// TIA Portal project "1905391_000_005" (V16)

(* hardware
DEVICE "S7-1200 station_1"  S7-1200 Station
   slot 0: "Rack_0"  S7-1200 Rack  Rack  V1.0
   slot 1: "PLC_1"  CPU 1211C DC/DC/DC  6ES7 211-1AE40-0XB0  V4.4
DEVICE "HMI_1"  TP900 Comfort
   slot 0: "HMI_1"  TP900 Comfort  6AV2 124-0JC01-0AX0  16.0.0.0
   slot 1: "HMI_RT_1"  TP900 Comfort  6AV2 124-0JC01-0AX0  16.0.0.0
   slot 5: "HMI_1.IE_CP_1"  PROFINET Interface  16.0.0.0
      slot 1: "PROFINET Interface_1"  PROFINET Interface
         slot 1: "Port_1"  Port
         slot 2: "Port_2"  Port
   slot 7: "HMI_1.MPI/DP_CP_1"  MPI/DP Interface  16.0.0.0
*)

// ===== PLC "PLC_1"  CPU 1211C DC/DC/DC =====

VAR_GLOBAL   // PLC tag table "Default tag table"
   "System_Byte" AT %MB1 : Byte;
   "FirstScan" AT %M1.0 : Bool;
   "DiagStatusUpdate" AT %M1.1 : Bool;
   "AlwaysTRUE" AT %M1.2 : Bool;
   "AlwaysFALSE" AT %M1.3 : Bool;
   "Clock_Byte" AT %MB0 : Byte;
   "Clock_10Hz" AT %M0.0 : Bool;
   "Clock_5Hz" AT %M0.1 : Bool;
   "Clock_2.5Hz" AT %M0.2 : Bool;
   "Clock_2Hz" AT %M0.3 : Bool;
   "Clock_1.25Hz" AT %M0.4 : Bool;
   "Clock_1Hz" AT %M0.5 : Bool;
   "Clock_0.625Hz" AT %M0.6 : Bool;
   "Clock_0.5Hz" AT %M0.7 : Bool;
END_VAR

VAR_GLOBAL CONSTANT   // PLC tag table "Default tag table"
   "STRING_LENGTH" : Int := 20;
   "ADP_PARAMETER_LENGTH" : Int := 5;
   "NULL_TOKEN" : Int := -1;
END_VAR

TYPE "Database.UDT"
   STRUCT
      elements : "Elements.Data.UDT";
      wires : "Wires.Data.UDT";
   END_STRUCT;
END_TYPE

TYPE "Divider.UDT"
   STRUCT
      background_animate : Int;
      background_visible : Bool;
      line_animate : Int;
      line_visible : Bool;
   END_STRUCT;
END_TYPE

TYPE "Row_Data.UDT"
   STRUCT
      background_animate : Int;
      background_visible : Bool;
      cell_0_animate : Int;
      cell_0_value : String[50];
      cell_0_visible : Bool;
      cell_1_animate : Int;
      cell_1_enable : Bool;
      cell_1_input_finished : Bool;
      cell_1_value : String[50];
      cell_1_visible : Bool;
   END_STRUCT;
END_TYPE

TYPE "Row_Label.UDT"
   STRUCT
      background_animate : Int;
      background_visible : Bool;
      cell_0_animate : Int;
      cell_0_value : String[50];
      cell_0_visible : Bool;
      cell_1_animate : Int;
      cell_1_value : String[50];
      cell_1_visible : Bool;
   END_STRUCT;
END_TYPE

TYPE "HMI_Interface.UDT"
   STRUCT
      elements : "Elements.HMI.UDT";
      wires : "Wires.HMI.UDT";
   END_STRUCT;
END_TYPE

TYPE "LED_Interface.UDT"
   STRUCT
      elements : "Elements.LED.UDT";
      wires : "Wires.LED.UDT";
   END_STRUCT;
END_TYPE

TYPE "Navigation.UDT"
   STRUCT
      material_actuate : Bool;
      material_animate : Int;
      material_cover_visible : Bool;
      wire_actuate : Bool;
      wire_animate : Int;
      wire_cover_visible : Bool;
   END_STRUCT;
END_TYPE

TYPE "Row_Custom.UDT"
   STRUCT
      background_animate : Int;
      background_visible : Bool;
      cell_0_animate : Int;
      cell_0_enable : Bool;
      cell_0_input_finished : Bool;
      cell_0_value : String[50];
      cell_0_visible : Bool;
      cell_1_animate : Int;
      cell_1_enable : Bool;
      cell_1_input_finished : Bool;
      cell_1_value : String[50];
      cell_1_visible : Bool;
   END_STRUCT;
END_TYPE

// folder: ADP Data

TYPE "ADP.Row.2_Cells.UDT"
   STRUCT
      me : Array[0..1] of "ADP.Cell.UDT";
   END_STRUCT;
END_TYPE

TYPE "ADP.Cell.UDT"
   STRUCT
      color : String["ADP_PARAMETER_LENGTH"];
      flashing : String["ADP_PARAMETER_LENGTH"];
      h_align : String["ADP_PARAMETER_LENGTH"];
      lince_control : String["ADP_PARAMETER_LENGTH"];
      scroll_speed : String["ADP_PARAMETER_LENGTH"];
      size_and_face : String["ADP_PARAMETER_LENGTH"];
      v_align : String["ADP_PARAMETER_LENGTH"];
      value : String["STRING_LENGTH"];
   END_STRUCT;
END_TYPE

TYPE "ADP.Message_Buffer.UDT"
   STRUCT
      me : Array[0..999] of Byte;
   END_STRUCT;
END_TYPE

TYPE "ADP.Decoded.UDT"
   STRUCT
      color : "ADP.Decoded.Color.UDT";
      flash : "ADP.Decoded.Flash.UDT";
      horizontal_alignment : "ADP.Decoded.Horizontal_Alignment.UDT";
      line_control : "ADP.Decoded.Line_Control.UDT";
      scroll_speed : "ADP.Decoded.Scroll_Speed.UDT";
      size_and_face : "ADP.Decoded.Size_and_Face.UDT";
      vertical_alignment : "ADP.Decoded.Vertical_Alignment.UDT";
   END_STRUCT;
END_TYPE

TYPE "ADP.Decoded.Color.UDT"
   STRUCT
      black : String[8] := 'black';
      blue : String[8] := 'blue';
      green : String[8] := 'green';
      mix_1 : String[8] := 'mix 1';
      mix_2 : String[8] := 'mix 2';
      mix_3 : String[8] := 'mix 3';
      mix_4 : String[8] := 'mix 4';
      red : String[8] := 'red';
      white : String[8] := 'white';
      yellow : String[8] := 'yellow';
   END_STRUCT;
END_TYPE

TYPE "ADP.Decoded.Flash.UDT"
   STRUCT
      off : String[8] := 'off';
      on : String[8] := 'on';
   END_STRUCT;
END_TYPE

TYPE "ADP.Decoded.Horizontal_Alignment.UDT"
   STRUCT
      center : String[8] := 'center';
      left : String[8] := 'left';
      right : String[8] := 'right';
   END_STRUCT;
END_TYPE

TYPE "ADP.Encoded.UDT"
VERSION : 0.1
   STRUCT
      file_system : "ADP.Encoded.File_System.UDT";
      formatting : "ADP.Encoded.Formatting.UDT";
   END_STRUCT;
END_TYPE

TYPE "ADP.Message_Formats.Encoded.UDT"
   STRUCT
      color : String [5];
      flash : String [5];
      scroll_speed : String [5];
      size_and_face : String [5];
      vertical_alignment : String [5];
      horizontal_alignment : String [5];
   END_STRUCT;
END_TYPE

TYPE "ADP.Message_Formats.Decoded.UDT"
   STRUCT
      color : String [20];
      flash : String [20];
      scroll_speed : String [20];
      size_and_face : String [20];
      vertical_alignment : String [20];
      horizontal_alignment : String [20];
   END_STRUCT;
END_TYPE

TYPE "ADP.Decoded.Scroll_Speed.UDT"
   STRUCT
      slowest : String[9] := 'slowest';
      slow : String[9] := 'slow';
      normal : String[9] := 'normal';
      fast : String[9] := 'fast';
      fastest : String[9] := 'fastest';
   END_STRUCT;
END_TYPE

TYPE "ADP.Decoded.Size_and_Face.UDT"
   STRUCT
      bold_5 : String[11] := 'bold 5';
      bold_11 : String[11] := 'bold 11';
      bold_14 : String[11] := 'bold 14';
      bold_15 : String[11] := 'bold 15';
      bold_16 : String[11] := 'bold 16';
      bold_22 : String[11] := 'bold 22';
      bold_30 : String[11] := 'bold 30';
      bold_32 : String[11] := 'bold 32';
      bold_40 : String[11] := 'bold 40';
      normal_5 : String[11] := 'normal 5';
      normal_7 : String[11] := 'normal 7';
      normal_9 : String[11] := 'normal 9';
      normal_11 : String[11] := 'normal 11';
      normal_14 : String[11] := 'normal 14';
      normal_15 : String[11] := 'normal 15';
      normal_16 : String[11] := 'normal 16';
      normal_22 : String[11] := 'normal 22';
      normal_24 : String[11] := 'normal 24';
      normal_30 : String[11] := 'normal 30';
      normal_32 : String[11] := 'normal 32';
      normal_40 : String[11] := 'normal 40';
   END_STRUCT;
END_TYPE

TYPE "ADP.Decoded.Vertical_Alignment.UDT"
   STRUCT
      bottom_hold : String[15] := 'bottom hold';
      fill_hold : String[15] := 'fill hold';
      middle_hold : String[15] := 'middle hold';
      top_hold : String[15] := 'top hold';
      bottom_scroll : String[15] := 'bottom scroll';
      fill_scroll : String[15] := 'fill scroll';
      middle_scroll : String[15] := 'middle scroll';
      top_scroll : String[15] := 'top scroll';
   END_STRUCT;
END_TYPE

TYPE "ADP.Encoded.File_System.UDT"
   STRUCT
      "00 Start of Header" : String[5] := '$01';
      "01 Address" : String[5] := 'Z00';
      "02 Start of Text" : String[5] := '$02';
      "03 Command & File" : String[5] := 'AA';
      "04 END" : String[5] := '$04';
   END_STRUCT;
END_TYPE

TYPE "ADP.Encoded.Formatting.UDT"
   STRUCT
      color : "ADP.Encoded.Formatting.Color.UDT";
      flashing : "ADP.Encoded.Formatting.Flashing.UDT";
      horizontal_alignment : "ADP.Encoded.Formatting.Horizonta_Alignment.UDT";
      line_control : "ADP.Encoded.Formatting.Line_Control.UDT";
      scroll_speed : "ADP.Encoded.Formatting.Scroll_Speed.UDT";
      size_and_face : "ADP.Encoded.Formatting.Size_and_Face.UDT";
      vertical_alignment : "ADP.Encoded.Formatting.Vertical_Alignment.UDT";
   END_STRUCT;
END_TYPE

TYPE "ADP.Encoded.Formatting.Color.UDT"
   STRUCT
      black : String[5] := '$1C0';
      blue : String[5] := '$1C8';
      green : String[5] := '$1C2';
      mix_1 : String[5] := '$1C4';
      mix_2 : String[5] := '$1C5';
      mix_3 : String[5] := '$1C6';
      mix_4 : String[5] := '$1CY';
      red : String[5] := '$1C1';
      white : String[5] := '$1C9';
      yellow : String[5] := '$1C3';
   END_STRUCT;
END_TYPE

TYPE "ADP.Encoded.Formatting.Flashing.UDT"
   STRUCT
      off : String[5] := '$070';
      on : String[5] := '$071';
   END_STRUCT;
END_TYPE

TYPE "ADP.Encoded.Formatting.Size_and_Face.UDT"
   STRUCT
      bold_5 : String[5] := '$1AG';
      bold_11 : String[5] := '$1AH';
      bold_14 : String[5] := '$1A5';
      bold_15 : String[5] := '$1A6';
      bold_16 : String[5] := '$1A7';
      bold_22 : String[5] := '$1AC';
      bold_30 : String[5] := '$1AI';
      bold_32 : String[5] := '$1AJ';
      bold_40 : String[5] := '$1AK';
      normal_5 : String[5] := '$1A0';
      normal_7 : String[5] := '$1A1';
      normal_9 : String[5] := '$1A8';
      normal_11 : String[5] := '$1A9';
      normal_14 : String[5] := '$1A2';
      normal_15 : String[5] := '$1A3';
      normal_16 : String[5] := '$1A4';
      normal_22 : String[5] := '$1AA';
      normal_24 : String[5] := '$1AB';
      normal_30 : String[5] := '$1AD';
      normal_32 : String[5] := '$1AE';
      normal_40 : String[5] := '$1AF';
   END_STRUCT;
END_TYPE

TYPE "ADP.Encoded.Formatting.Horizonta_Alignment.UDT"
   STRUCT
      center : String[5] := '$L1';
      left : String[5] := '$L0';
      right : String[5] := '$L2';
   END_STRUCT;
END_TYPE

TYPE "ADP.Encoded.Formatting.Vertical_Alignment.UDT"
   STRUCT
      middle_hold : String[5] := '$1B b';
      fill_hold : String[5] := '$1B"b';
      bottom_hold : String[5] := '$1B&b';
      top_hold : String[5] := '$1B0b';
      bottom_scroll : String[5] := '$1B a';
      fill_scroll : String[5] := '$1B"a';
      middle_scroll : String[5] := '$1B&a';
      top_scroll : String[5] := '$1B0a';
   END_STRUCT;
END_TYPE

TYPE "ADP.Encoded.Formatting.Scroll_Speed.UDT"
   STRUCT
      slowest : String[5] := '$15';
      slow : String[5] := '$16';
      normal : String[5] := '$17';
      fast : String[5] := '$18';
      fastest : String[5] := '$19';
   END_STRUCT;
END_TYPE

TYPE "ADP.Encoded.Formatting.Line_Control.UDT"
   STRUCT
      new_line : String[5] := '$R';
      word_wrap : String[5] := '';
   END_STRUCT;
END_TYPE

TYPE "ADP.Decoded.Line_Control.UDT"
   STRUCT
      new_line : String[9] := 'new line';
      word_wrap : String[9] := 'word wrap';
   END_STRUCT;
END_TYPE

// folder: Element Data

TYPE "Elements.HMI.UDT"
   STRUCT
      chromium : "Row.(IOF.String_IOF.Real).UDT";
      custom : "Row.(IOF.String_IOF.Real).UDT";
      header : "Row.(IOF.String_IOF.String).UDT";
      heat : "Row.(IOF.String_IOF.Real).UDT";
      manganese : "Row.(IOF.String_IOF.Real).UDT";
      molybdenum : "Row.(IOF.String_IOF.Real).UDT";
      nickel : "Row.(IOF.String_IOF.Real).UDT";
      silicon : "Row.(IOF.String_IOF.Real).UDT";
      vanadium : "Row.(IOF.String_IOF.Real).UDT";
   END_STRUCT;
   // header.cell_00.value := 'Material';
   // header.cell_01.value := 'Bags';
END_TYPE

TYPE "Elements.Data.UDT"
   STRUCT
      chromium : Real;
      custom_value : Real;
      custom_name : String[50];
      heat : Real;
      manganese : Real;
      molybdenum : Real;
      nickel : Real;
      silicon : Real;
      vanadium : Real;
   END_STRUCT;
END_TYPE

TYPE "Elements.LED.UDT"
   STRUCT
      chromium : "ADP.Row.2_Cells.UDT";
      custom : "ADP.Row.2_Cells.UDT";
      header : "ADP.Row.2_Cells.UDT";
      heat : "ADP.Row.2_Cells.UDT";
      manganese : "ADP.Row.2_Cells.UDT";
      molybdenum : "ADP.Row.2_Cells.UDT";
      nickel : "ADP.Row.2_Cells.UDT";
      silicon : "ADP.Row.2_Cells.UDT";
      vanadium : "ADP.Row.2_Cells.UDT";
   END_STRUCT;
   // chromium.me[0].value := 'chromium';
   // heat.me[0].value := 'heat';
   // manganese.me[0].value := 'manganese';
   // molybdenum.me[0].value := 'molybdenum';
   // nickel.me[0].value := 'nickel';
   // silicon.me[0].value := 'silicon';
   // vanadium.me[0].value := 'vanadium';
   // custom.me[0].value := 'Custom';
   // header.me[0].value := 'Material';
   // header.me[1].value := 'Bags';
END_TYPE

// folder: Wire Data

TYPE "Wire.UDT"
   STRUCT
      aluminum : Real;
      calcium_silicon : Real;
      carbon : Real;
      custom : Real;
      heat : Real;
      sulfur : Real;
   END_STRUCT;
END_TYPE

TYPE "Wires.LED.UDT"
   STRUCT
      aluminum : "ADP.Row.2_Cells.UDT";
      calcium_silicon : "ADP.Row.2_Cells.UDT";
      carbon : "ADP.Row.2_Cells.UDT";
      custom : "ADP.Row.2_Cells.UDT";
      heat : "ADP.Row.2_Cells.UDT";
      sulfur : "ADP.Row.2_Cells.UDT";
   END_STRUCT;
   // aluminum.me[0].value := 'AL Wire';
   // calcium_silicon.me[0].value := 'Cal/Sil Wire';
   // carbon.me[0].value := 'Carbon Wire';
   // heat.me[0].value := 'HEAT';
   // sulfur.me[0].value := 'Sulfur Wire';
   // custom.me[0].value := 'Custom';
END_TYPE

TYPE "Wire.HMI.UDT"
   STRUCT
      aluminum : "Row_Data.UDT";
      bottom_border : "Divider.UDT";
      calcium_silicon : "Row_Data.UDT";
      carbon : "Row_Data.UDT";
      divider : "Divider.UDT";
      header : "Row_Data.UDT";
      heat : "Row_Data.UDT";
      sulfur : "Row_Data.UDT";
   END_STRUCT;
END_TYPE

// folder: data

DATA_BLOCK "Database.Data"   // DB1
{ S7_Optimized_Access := 'TRUE' }
VERSION : 0.1
BEGIN
END_DATA_BLOCK

// folder: display/HMI

DATA_BLOCK "HMI_Interface.Data"   // DB2
{ S7_Optimized_Access := 'TRUE' }
VERSION : 0.1
BEGIN
END_DATA_BLOCK

// folder: display/LED

DATA_BLOCK "LED_Interface.Data"   // DB3
{ S7_Optimized_Access := 'TRUE' }
VERSION : 0.1
BEGIN
END_DATA_BLOCK

// folder: (top level)

FUNCTION "Row_Data.Background.Animate" : Void   // FC1, SCL
{ S7_Optimized_Access := 'TRUE' }
VERSION : 0.1
   VAR_IN_OUT
      background : Int;
   END_VAR
BEGIN
END_FUNCTION

FUNCTION "Strip_Sign" : String   // FC20, SCL
{ S7_Optimized_Access := 'TRUE' }
VERSION : 0.1
   VAR_INPUT
      "string" : String;
   END_VAR
   VAR_TEMP
      Length : Int;
      "String Box" : String;
      "Test Character" : String;
   END_VAR
   VAR CONSTANT
      "+" : Char := '+';
      "-" : Char := '-';
   END_VAR
BEGIN
   #"String Box" := #string;
   #"Test Character" := LEFT_STRING(IN := #"String Box",
                                    L := 1);
   IF #"Test Character" = #"+" OR #"Test Character" = #"-" THEN
       #Length := LEN(#"String Box");
       #"String Box" := RIGHT_STRING(IN := #"String Box", L := #Length - 1);

   END_IF;
   #"Strip Sign" := #"String Box";
END_FUNCTION

FUNCTION "Trim" : String   // FC21, SCL
{ S7_Optimized_Access := 'TRUE' }
AUTHOR : Machado
FAMILY : String
VERSION : 1.0
// removes leading and trailing whitespace from input string
   VAR_INPUT
      "string" : String;
   END_VAR
   VAR_TEMP
      ret : String;
   END_VAR
   VAR CONSTANT
      space : String := ' ';
   END_VAR
BEGIN
   #ret := #string;
   WHILE LEFT(IN := #ret, L := 1) = #space DO
       #ret := RIGHT(IN := #ret, L := LEN(#ret) - 1);
   END_WHILE;
   WHILE RIGHT(IN := #ret, L := 1) = #space DO
       #ret := LEFT(IN := #ret, L := LEN(#ret) - 1);
   END_WHILE;
   #Trim := #ret;
END_FUNCTION

FUNCTION "Upper" : String   // FC22, SCL
{ S7_Optimized_Access := 'TRUE' }
AUTHOR : Machado
FAMILY : String
VERSION : 1.0
// returns the input string converted to all upper case
   VAR_INPUT
      "string" : String;
   END_VAR
   VAR_TEMP
      "type" : Bool;
      stringBox : String;
      status : Int;
      charArr : Array[0..255] of Char;
      cntChar : UInt;
      pChar : Int;
   END_VAR
   VAR CONSTANT
      asciiLow : Char := 'a';
      asciiHigh : Char := 'z';
      asciiCaseOffset : Int := 32;
   END_VAR
BEGIN
   Strg_TO_Chars(Strg := #string,
                 pChars := 0,
                 Cnt => #cntChar,
                 Chars := #charArr);

   FOR #pChar := 0 TO UINT_TO_INT(#cntChar) - 1 DO
       IF #asciiLow <= #charArr[#pChar] AND #charArr[#pChar] <= #asciiHigh THEN
           #charArr[#pChar] := INT_TO_CHAR(CHAR_TO_INT(#charArr[#pChar]) - #asciiCaseOffset);
       END_IF;
   END_FOR;

   Chars_TO_Strg(Chars := #charArr,
                 pChars := 0,
                 Cnt := #cntChar,
                 Strg => #stringBox);

   #Upper := #stringBox;
END_FUNCTION

ORGANIZATION_BLOCK "Main"   // OB1, LAD, ProgramCycle
TITLE = "Main Program Sweep (Cycle)"
{ S7_Optimized_Access := 'TRUE' }
VERSION : 0.1
   VAR_INPUT
      Initial_Call : Bool;   // Initial call of this OB
      Remanence : Bool;   // =True, if remanent data are available
   END_VAR
BEGIN
END_ORGANIZATION_BLOCK

// folder: display

FUNCTION_BLOCK "Display"   // FB5, SCL
{ S7_Optimized_Access := 'TRUE' }
VERSION : 0.1
BEGIN
   REGION "HMI"

   END_REGION

   REGION "LED"

   END_REGION
END_FUNCTION_BLOCK

// folder: display/HMI

FUNCTION_BLOCK "HMI"   // FB6, SCL
{ S7_Optimized_Access := 'TRUE' }
VERSION : 0.1
   VAR_IN_OUT
      interface : "HMI_Interface.UDT";
   END_VAR
   VAR
      place_holder : Bool;
   END_VAR
BEGIN
   REGION "VALIDATE INPUT"
       "HMI.Validate"();
   END_REGION


   REGION "DISPLAY VALUES"
       // may not be needed, handeled entirely in middleware
   END_REGION


   REGION "ANIMATE"
       "HMI.Animate"();
   END_REGION
END_FUNCTION_BLOCK

FUNCTION "HMI.Animate" : Void   // FC8, SCL
{ S7_Optimized_Access := 'TRUE' }
VERSION : 0.1
BEGIN
   "Element.Animate"();
   "Wire.Animate"();
END_FUNCTION

FUNCTION "HMI.Validate" : Void   // FC9, SCL
{ S7_Optimized_Access := 'TRUE' }
VERSION : 0.1
BEGIN
   "Element.Validate"();
   "Wire.Validate"();
END_FUNCTION

FUNCTION "HMI.Display" : Void   // FC10, SCL
{ S7_Optimized_Access := 'TRUE' }
VERSION : 0.1
   VAR_INPUT
      database : Bool;
   END_VAR
BEGIN
END_FUNCTION

// folder: display/HMI/Wire

FUNCTION "HMI.Animate.Wire" : Void   // FC3, SCL
{ S7_Optimized_Access := 'TRUE' }
VERSION : 0.1
   VAR_IN_OUT
      wire : "Wire.HMI.UDT";
   END_VAR
BEGIN
END_FUNCTION

FUNCTION "Wire.Animate.Aluminum" : Void   // FC4, SCL
{ S7_Optimized_Access := 'TRUE' }
VERSION : 0.1
BEGIN
END_FUNCTION

// folder: display/LED

FUNCTION_BLOCK "LED"   // FB7, SCL
{ S7_Optimized_Access := 'TRUE' }
VERSION : 0.1
   VAR
      Elements_Sign : "Elements_Sign";
      Wires_Sign : "Wires_Sign";
   END_VAR
BEGIN
   REGION "ELEMENTS"
       #Elements_Sign();
   END_REGION

   REGION "WIRES"
       #Wires_Sign();
   END_REGION
END_FUNCTION_BLOCK

FUNCTION_BLOCK "LED.Sign.Send"   // FB9, SCL
{ S7_Optimized_Access := 'TRUE' }
VERSION : 0.1
   VAR_INPUT
      data : "ADP.Message_Buffer.UDT";
      id : Conn_Ouc;
      request : Bool;
   END_VAR
   VAR
      TSEND : TSEND;
   END_VAR
BEGIN
   #TSEND(REQ := #request,
          ID := #id,
          DATA := #data);
END_FUNCTION_BLOCK

FUNCTION_BLOCK "LED.Sign"   // FB10, SCL
{ S7_Optimized_Access := 'TRUE' }
VERSION : 0.1
   VAR_INPUT
      id : Conn_Ouc;
      connection_parameters : TCON_Param;
      requests : Struct
         connect : Bool;
         diagnostics : Bool;
         disconnect : Bool;
         reset : Bool;
         send : Bool;
      END_STRUCT;
   END_VAR
   VAR
      Connect : "LED.Sign.Connect";
      Disconnect : "LED.Sign.Disconnect";
      Send : "LED.Sign.Send";
      Reset : "LED.Sign.Reset";
      Diagnostics : "LED.Sign.Diagnostics";
   END_VAR
BEGIN
   #Connect(request := #requests.connect,
            id := #id,
            connection_parameters := #connection_parameters);

   #Disconnect(id := #id,
               request := #requests.disconnect);

   #Send(id := #id,
         request := #requests.send);

   #Reset(id := #id,
          request := #requests.reset);

   #Diagnostics(id := #id,
                request := #requests.diagnostics);
END_FUNCTION_BLOCK

FUNCTION_BLOCK "LED.Sign.Connect"   // FB11, SCL
{ S7_Optimized_Access := 'TRUE' }
VERSION : 0.1
   VAR_INPUT
      request : Bool;
      id : Conn_Ouc;
      connection_parameters : TCON_Param;
   END_VAR
   VAR
      TCON : TCON;
   END_VAR
BEGIN
   #TCON(REQ := #request,
         ID := #id,
         CONNECT := #connection_parameters);
END_FUNCTION_BLOCK

FUNCTION_BLOCK "LED.Sign.Reset"   // FB12, SCL
{ S7_Optimized_Access := 'TRUE' }
VERSION : 0.1
   VAR_INPUT
      request : Bool;
      id : Conn_Ouc;
   END_VAR
   VAR
      T_RESET : T_RESET;
   END_VAR
BEGIN
   #T_RESET(REQ:=#request,
            ID:=#id,
            DONE=>_bool_out_,
            BUSY=>_bool_out_,
            ERROR=>_bool_out_,
            STATUS=>_word_out_);
END_FUNCTION_BLOCK

FUNCTION_BLOCK "LED.Sign.Disconnect"   // FB13, SCL
{ S7_Optimized_Access := 'TRUE' }
VERSION : 0.1
   VAR_INPUT
      request : Bool;
      id : Conn_Ouc;
   END_VAR
   VAR
      TDISCON : TDISCON;
   END_VAR
BEGIN
   #TDISCON(REQ := #request,
            ID := #id);
END_FUNCTION_BLOCK

FUNCTION_BLOCK "LED.Sign.Diagnostics"   // FB14, SCL
{ S7_Optimized_Access := 'TRUE' }
VERSION : 0.1
   VAR_INPUT
      request : Bool;
      id : Conn_Ouc;
   END_VAR
   VAR
      T_DIAG : T_DIAG;
   END_VAR
BEGIN
   #T_DIAG(REQ:=#request,
           ID:=#id);
END_FUNCTION_BLOCK

// folder: display/LED/Elements Sign

FUNCTION_BLOCK "Elements_Sign"   // FB16, SCL
{ S7_Optimized_Access := 'TRUE' }
VERSION : 0.1
   VAR
      Sign : "LED.Sign";
      id : Conn_Ouc;
      connection_parameters : TCON_Param;
   END_VAR
BEGIN
   "Elements_Sign.Assemble_Message"();
   #Sign(id := #id,
         connection_parameters := #connection_parameters);
END_FUNCTION_BLOCK

FUNCTION "Elements_Sign.Assemble_Message" : Void   // FC11, SCL
{ S7_Optimized_Access := 'TRUE' }
VERSION : 0.1
BEGIN
END_FUNCTION

// folder: display/LED/Wires Sign

FUNCTION_BLOCK "Wires_Sign"   // FB15, SCL
{ S7_Optimized_Access := 'TRUE' }
VERSION : 0.1
   VAR
      Sign : "LED.Sign";
      id : Conn_Ouc;
      connection_parameters : TCON_Param;
   END_VAR
BEGIN
   "Wires_Sign.Assemble_Message"();
   #Sign(id := #id,
         connection_parameters := #connection_parameters);
END_FUNCTION_BLOCK

FUNCTION "Wires_Sign.Assemble_Message" : Void   // FC12, SCL
{ S7_Optimized_Access := 'TRUE' }
VERSION : 0.1
BEGIN
END_FUNCTION

// folder: divider

FUNCTION "Divider.Show" : Void   // FC2, SCL
{ S7_Optimized_Access := 'TRUE' }
VERSION : 0.1
   VAR_IN_OUT
      divider : "Divider.UDT";
   END_VAR
   VAR CONSTANT
      MODE : Bool := TRUE;
   END_VAR
BEGIN
   #divider.background_visible := #MODE;
   #divider.line_visible := #MODE;
END_FUNCTION

FUNCTION "Divider.Hide" : Void   // FC2, SCL
{ S7_Optimized_Access := 'TRUE' }
VERSION : 0.1
   VAR_IN_OUT
      divider : "Divider.UDT";
   END_VAR
   VAR CONSTANT
      MODE : Bool := FALSE;
   END_VAR
BEGIN
   #divider.background_visible := #MODE;
   #divider.line_visible := #MODE;
END_FUNCTION

FUNCTION "Divider.Hide_Line" : Void   // FC13, SCL
{ S7_Optimized_Access := 'TRUE' }
VERSION : 0.1
   VAR_TEMP
      divider : "Divider.UDT";
   END_VAR
   VAR CONSTANT
      MODE : Bool := TRUE;
   END_VAR
BEGIN
   #divider.line_visible := #MODE;
END_FUNCTION

// folder: middleware

FUNCTION_BLOCK "Middleware"   // FB2, SCL
{ S7_Optimized_Access := 'TRUE' }
VERSION : 0.1
   VAR_IN_OUT
      database : "Database.UDT";
      hmi : "HMI_Interface.UDT";
      led : "LED_Interface.UDT";
   END_VAR
   VAR
      elements : "Elements";
      wires : "Wires";
   END_VAR
BEGIN
   #elements(database := #database.elements,
             hmi := #hmi.elements,
             led := #led.elements);

   #wires(database := #database.wires,
          hmi := #hmi.wires,
          led := #led.wires);
END_FUNCTION_BLOCK

// folder: row_data

FUNCTION "Row_Data.Animate" : Void   // FC5, SCL
{ S7_Optimized_Access := 'TRUE' }
VERSION : 0.1
   VAR_IN_OUT
      row_data : "Row_Data.UDT";
   END_VAR
BEGIN
   #row_data.background_animate := "NULL_TOKEN";
   #row_data.cell_0_animate := "NULL_TOKEN";
   #row_data.cell_1_animate := "NULL_TOKEN";
END_FUNCTION

FUNCTION "Row_Data.Show" : Void   // FC6, SCL
{ S7_Optimized_Access := 'TRUE' }
VERSION : 0.1
   VAR_IN_OUT
      row_data : "Row_Data.UDT";
   END_VAR
   VAR CONSTANT
      MODE : Bool := TRUE;
   END_VAR
BEGIN
   #row_data.background_visible := #MODE;
   #row_data.cell_0_visible := #MODE;
   #row_data.cell_1_visible := #MODE;
END_FUNCTION

FUNCTION "Row_Data.Hide" : Void   // FC6, SCL
{ S7_Optimized_Access := 'TRUE' }
VERSION : 0.1
   VAR_IN_OUT
      row_data : "Row_Data.UDT";
   END_VAR
   VAR CONSTANT
      MODE : Bool := FALSE;
   END_VAR
BEGIN
   #row_data.background_visible := #MODE;
   #row_data.cell_0_visible := #MODE;
   #row_data.cell_1_visible := #MODE;
END_FUNCTION

FUNCTION "Row_Data.Enable" : Void   // FC7, SCL
{ S7_Optimized_Access := 'TRUE' }
VERSION : 0.1
   VAR_IN_OUT
      row_data : "Row_Data.UDT";
   END_VAR
BEGIN
   #row_data.cell_1_enable := TRUE;
END_FUNCTION

// ===== library types =====

TYPE "Row.UDT"
   STRUCT
      background_animate : Int;
      background_visible : Bool;
      cell_0_animate : Int;
      cell_0_value : String[50];
      cell_0_visible : Bool;
      cell_1_animate : Int;
      cell_1_enable : Bool;
      cell_1_input_finished : Bool;
      cell_1_value : String[50];
      cell_1_visible : Bool;
   END_STRUCT;
END_TYPE

// ===== library: MasterCopy "Copy of PLC data types in ADP Data" =====

// folder: ADP Data

TYPE "ADP: Encoded"
VERSION : 0.1
   STRUCT
      file_system : "ADP: Encoded: File System";
      formatting : "ADP: Encoded: Formatting";
   END_STRUCT;
END_TYPE

TYPE "ADP: Decoded"
   STRUCT
      color : "ADP: Decoded: Color";
      flash : "ADP: Decoded: Flash";
      horizontal_alignment : "ADP: Decoded: Horizontal Alignment";
      line_control : "ADP: Decoded: Line Control";
      scroll_speed : "ADP: Decoded: Scroll Speed";
      size_and_face : "ADP: Decoded: Size and Face";
      vertical_alignment : "ADP: Decoded: Vertical Alignment";
   END_STRUCT;
END_TYPE

TYPE "ADP: Decoded: Color"
   STRUCT
      black : String[8] := 'black';
      blue : String[8] := 'blue';
      green : String[8] := 'green';
      mix_1 : String[8] := 'mix 1';
      mix_2 : String[8] := 'mix 2';
      mix_3 : String[8] := 'mix 3';
      mix_4 : String[8] := 'mix 4';
      red : String[8] := 'red';
      white : String[8] := 'white';
      yellow : String[8] := 'yellow';
   END_STRUCT;
END_TYPE

TYPE "ADP: Decoded: Flash"
   STRUCT
      off : String[8] := 'off';
      on : String[8] := 'on';
   END_STRUCT;
END_TYPE

TYPE "ADP: Decoded: Horizontal Alignment"
   STRUCT
      center : String[8] := 'center';
      left : String[8] := 'left';
      right : String[8] := 'right';
   END_STRUCT;
END_TYPE

TYPE "ADP: Message Formats: Encoded"
   STRUCT
      color : String [5];
      flash : String [5];
      scroll_speed : String [5];
      size_and_face : String [5];
      vertical_alignment : String [5];
      horizontal_alignment : String [5];
   END_STRUCT;
END_TYPE

TYPE "ADP: Message Formats: Decoded"
   STRUCT
      color : String [20];
      flash : String [20];
      scroll_speed : String [20];
      size_and_face : String [20];
      vertical_alignment : String [20];
      horizontal_alignment : String [20];
   END_STRUCT;
END_TYPE

TYPE "ADP: Decoded: Scroll Speed"
   STRUCT
      slowest : String[9] := 'slowest';
      slow : String[9] := 'slow';
      normal : String[9] := 'normal';
      fast : String[9] := 'fast';
      fastest : String[9] := 'fastest';
   END_STRUCT;
END_TYPE

TYPE "ADP: Decoded: Size and Face"
   STRUCT
      bold_5 : String[11] := 'bold 5';
      bold_11 : String[11] := 'bold 11';
      bold_14 : String[11] := 'bold 14';
      bold_15 : String[11] := 'bold 15';
      bold_16 : String[11] := 'bold 16';
      bold_22 : String[11] := 'bold 22';
      bold_30 : String[11] := 'bold 30';
      bold_32 : String[11] := 'bold 32';
      bold_40 : String[11] := 'bold 40';
      normal_5 : String[11] := 'normal 5';
      normal_7 : String[11] := 'normal 7';
      normal_9 : String[11] := 'normal 9';
      normal_11 : String[11] := 'normal 11';
      normal_14 : String[11] := 'normal 14';
      normal_15 : String[11] := 'normal 15';
      normal_16 : String[11] := 'normal 16';
      normal_22 : String[11] := 'normal 22';
      normal_24 : String[11] := 'normal 24';
      normal_30 : String[11] := 'normal 30';
      normal_32 : String[11] := 'normal 32';
      normal_40 : String[11] := 'normal 40';
   END_STRUCT;
END_TYPE

TYPE "ADP: Decoded: Vertical Alignment"
   STRUCT
      bottom_hold : String[15] := 'bottom hold';
      fill_hold : String[15] := 'fill hold';
      middle_hold : String[15] := 'middle hold';
      top_hold : String[15] := 'top hold';
      bottom_scroll : String[15] := 'bottom scroll';
      fill_scroll : String[15] := 'fill scroll';
      middle_scroll : String[15] := 'middle scroll';
      top_scroll : String[15] := 'top scroll';
   END_STRUCT;
END_TYPE

TYPE "ADP: Encoded: File System"
   STRUCT
      "00 Start of Header" : String[5] := '$01';
      "01 Address" : String[5] := 'Z00';
      "02 Start of Text" : String[5] := '$02';
      "03 Command & File" : String[5] := 'AA';
      "04 END" : String[5] := '$04';
   END_STRUCT;
END_TYPE

TYPE "ADP: Encoded: Formatting"
   STRUCT
      color : "ADP: Encoded: Formatting: Color";
      flashing : "ADP: Encoded: Formatting: Flashing";
      horizontal_alignment : "ADP: Encoded: Formatting: Horizontal Alignment";
      line_control : "ADP: Encoded: Formatting: Line Control";
      scroll_speed : "ADP: Encoded: Formatting: Scroll Speed";
      size_and_face : "ADP: Encoded: Formatting: Size and Face";
      vertical_alignment : "ADP: Encoded: Formatting: Vertical Alignment";
   END_STRUCT;
END_TYPE

TYPE "ADP: Encoded: Formatting: Color"
   STRUCT
      black : String[5] := '$1C0';
      blue : String[5] := '$1C8';
      green : String[5] := '$1C2';
      mix_1 : String[5] := '$1C4';
      mix_2 : String[5] := '$1C5';
      mix_3 : String[5] := '$1C6';
      mix_4 : String[5] := '$1CY';
      red : String[5] := '$1C1';
      white : String[5] := '$1C9';
      yellow : String[5] := '$1C3';
   END_STRUCT;
END_TYPE

TYPE "ADP: Encoded: Formatting: Flashing"
   STRUCT
      off : String[5] := '$070';
      on : String[5] := '$071';
   END_STRUCT;
END_TYPE

TYPE "ADP: Encoded: Formatting: Size and Face"
   STRUCT
      bold_5 : String[5] := '$1AG';
      bold_11 : String[5] := '$1AH';
      bold_14 : String[5] := '$1A5';
      bold_15 : String[5] := '$1A6';
      bold_16 : String[5] := '$1A7';
      bold_22 : String[5] := '$1AC';
      bold_30 : String[5] := '$1AI';
      bold_32 : String[5] := '$1AJ';
      bold_40 : String[5] := '$1AK';
      normal_5 : String[5] := '$1A0';
      normal_7 : String[5] := '$1A1';
      normal_9 : String[5] := '$1A8';
      normal_11 : String[5] := '$1A9';
      normal_14 : String[5] := '$1A2';
      normal_15 : String[5] := '$1A3';
      normal_16 : String[5] := '$1A4';
      normal_22 : String[5] := '$1AA';
      normal_24 : String[5] := '$1AB';
      normal_30 : String[5] := '$1AD';
      normal_32 : String[5] := '$1AE';
      normal_40 : String[5] := '$1AF';
   END_STRUCT;
END_TYPE

TYPE "ADP: Encoded: Formatting: Horizontal Alignment"
   STRUCT
      center : String[5] := '$L1';
      left : String[5] := '$L0';
      right : String[5] := '$L2';
   END_STRUCT;
END_TYPE

TYPE "ADP: Encoded: Formatting: Vertical Alignment"
   STRUCT
      middle_hold : String[5] := '$1B b';
      fill_hold : String[5] := '$1B"b';
      bottom_hold : String[5] := '$1B&b';
      top_hold : String[5] := '$1B0b';
      bottom_scroll : String[5] := '$1B a';
      fill_scroll : String[5] := '$1B"a';
      middle_scroll : String[5] := '$1B&a';
      top_scroll : String[5] := '$1B0a';
   END_STRUCT;
END_TYPE

TYPE "ADP: Encoded: Formatting: Scroll Speed"
   STRUCT
      slowest : String[5] := '$15';
      slow : String[5] := '$16';
      normal : String[5] := '$17';
      fast : String[5] := '$18';
      fastest : String[5] := '$19';
   END_STRUCT;
END_TYPE

TYPE "ADP: Encoded: Formatting: Line Control"
   STRUCT
      new_line : String[5] := '$R';
      word_wrap : String[5] := '';
   END_STRUCT;
END_TYPE

TYPE "ADP: Decoded: Line Control"
   STRUCT
      new_line : String[9] := 'new line';
      word_wrap : String[9] := 'word wrap';
   END_STRUCT;
END_TYPE

(* ===== HMI "HMI_RT_1" =====
connection "HMI_Connection_1": ETHERNET, S7_1200_OMS

HMI tags "Default tag table"
   "Clock_Byte" : Byte = PLC Clock_Byte AT %MB0, 1 s

Template "Navigation" 800x480
   ScreenModuleView "Navigation_1" at 0,0 size 800x65; ScreenModuleType ""

screen "01 Wires" 800x480, template "Navigation"
   ScreenModuleView "heat" at 100,75 size 600x65; ScreenModuleType ""; Guid_{11997190-6447} 'HEAT'
   ScreenModuleView "label" at 100,140 size 600x65; ScreenModuleType ""
   ScreenModuleView "divider" at 100,205 size 600x5; ScreenModuleType ""
   ScreenModuleView "carbon" at 100,210 size 600x65; ScreenModuleType ""; Guid_{11997190-6447} 'CARBON'
   ScreenModuleView "calcium_silicon" at 100,275 size 600x65; ScreenModuleType ""; Guid_{11997190-6447} 'CAL/SIL'
   ScreenModuleView "aluminium" at 100,340 size 600x65; ScreenModuleType ""; Guid_{11997190-6447} 'ALUMINIUM'
   ScreenModuleView "sulfur" at 100,405 size 600x65; Guid_{11997190-6447} 'SULFUR'; ScreenModuleType ""
   ScreenModuleView "bottom_border" at 100,470 size 600x5; ScreenModuleType ""

screen "02 Elements" 800x480, template "Navigation"
   ScreenModuleView "heat" at 100,83 size 600x40; ScreenModuleType ""; Guid_{11997190-6447} 'HEAT'
   ScreenModuleView "material_label" at 100,123 size 600x40; ScreenModuleType ""
   ScreenModuleView "divider" at 100,163 size 600x5; ScreenModuleType ""
   ScreenModuleView "manganese" at 100,168 size 600x40; Guid_{11997190-6447} 'MANGANESE'; ScreenModuleType ""
   ScreenModuleView "silicon" at 100,208 size 600x40; Guid_{11997190-6447} 'SILICON'; ScreenModuleType ""
   ScreenModuleView "chromium" at 100,248 size 600x40; Guid_{11997190-6447} 'CHROMIUM'; ScreenModuleType ""
   ScreenModuleView "vanadium" at 100,288 size 600x40; Guid_{11997190-6447} 'VANADIUM'; ScreenModuleType ""
   ScreenModuleView "nickel" at 100,328 size 600x40; Guid_{11997190-6447} 'NICKEL'; ScreenModuleType ""
   ScreenModuleView "molybdenum" at 100,368 size 600x40; Guid_{11997190-6447} 'MOLYBDENUM'; ScreenModuleType ""
   ScreenModuleView "bottom_border" at 100,448 size 600x5; ScreenModuleType ""
   ScreenModuleView "custom" at 100,408 size 600x40; ScreenModuleType ""
*)

(* ===== HMI "HMI_RT_1" =====
system functions are stored by id; their names below are inferred from use

ScreenModuleEditorView "Row_Wire" 400x50
   Rectangle "Border" at 0,0 size 400x50
      Appearance <- "interface.background_animate"
   IOField "IOF R0 C0" at 5,5 size 190x45; FormatPattern ????????????????????
      ProcessValue <- "text_label"
      Appearance <- "interface.cell_0_animate"
      ObjectEnable <- "interface.cell_0_enable"
      Visibility <- "interface.cell_0_visible"
   IOField "IOF R0 C1" at 200,5 size 195x45; FormatPattern 9999999
      on OnFinishInput: SetBit("interface.cell_1_input_finished")
      Visibility <- "interface.cell_1_visible"
      ObjectEnable <- "interface.cell_1_enable"
      Appearance <- "interface.cell_1_animate"
*)

(* ===== HMI "HMI_RT_1" =====
system functions are stored by id; their names below are inferred from use

ScreenModuleEditorView "Row_Wire" 400x50
   Rectangle "Border" at 0,0 size 400x50
      Appearance <- "interface.background_animate"
      Visibility <- "interface.background_visible"
   IOField "IOF R0 C0" at 5,5 size 190x45; FormatPattern ????????????????????
      Appearance <- "interface.cell_0_animate"
      ProcessValue <- "text_label"
      Visibility <- "interface.cell_0_visible"
      ObjectEnable <- "interface.cell_0_enable"
   IOField "IOF R0 C1" at 200,5 size 195x45; FormatPattern 9999999
      on OnFinishInput: SetBit("interface.cell_1_input_finished")
      Visibility <- "interface.cell_1_visible"
      Appearance <- "interface.cell_1_animate"
      ObjectEnable <- "interface.cell_1_enable"
*)

(* ===== HMI "HMI_RT_1" =====
system functions are stored by id; their names below are inferred from use

ScreenModuleEditorView "Row_Wire" 400x50
   Rectangle "Border" at 0,0 size 400x50
      Visibility <- "interface.background_visible"
      Appearance <- "interface.background_animate"
   IOField "IOF R0 C0" at 5,5 size 190x45; FormatPattern ????????????????????
      Appearance <- "interface.cell_0_animate"
      Visibility <- "interface.cell_0_visible"
      ObjectEnable <- "interface.cell_0_enable"
      ProcessValue <- "interface.cell_0_value"
   IOField "IOF R0 C1" at 200,5 size 195x45; FormatPattern 9999999
      on OnFinishInput: SetBit("interface.cell_1_input_finished")
      Visibility <- "interface.cell_1_visible"
      Appearance <- "interface.cell_1_animate"
      ObjectEnable <- "interface.cell_1_enable"
*)

(* ===== HMI "HMI_RT_1" =====
system functions are stored by id; their names below are inferred from use

ScreenModuleEditorView "Row_Wire" 400x50
   Rectangle "Border" at 0,0 size 400x50
      Visibility <- "interface.background_visible"
      Appearance <- "interface.background_animate"
   IOField "IOF R0 C0" at 5,5 size 190x45; FormatPattern ????????????????????
      Appearance <- "interface.cell_0_animate"
      Visibility <- "interface.cell_0_visible"
      ProcessValue <- "interface.cell_0_value"
      ObjectEnable <- "interface.cell_0_enable"
   IOField "IOF R0 C1" at 200,5 size 195x45; FormatPattern 9999999
      on OnFinishInput: SetBit("interface.cell_1_input_finished")
      Visibility <- "interface.cell_1_visible"
      Appearance <- "interface.cell_1_animate"
      ObjectEnable <- "interface.cell_1_enable"
*)

(* ===== HMI "HMI_RT_1" =====
system functions are stored by id; their names below are inferred from use

ScreenModuleEditorView "Row_Wire" 400x65
   Rectangle "Border" at 0,0 size 400x65
      Visibility <- "interface.background_visible"
      Appearance <- "interface.background_animate"
   TextField "TF R0 C0" at 5,5 size 190x60; Text 'Text'
      Visibility <- "interface.cell_0_visible"
   IOField "IOF R0 C1" at 200,5 size 195x60; FormatPattern 9999999
      on OnFinishInput: SetBit("interface.cell_1_input_finished")
      Visibility <- "interface.cell_1_visible"
      ObjectEnable <- "interface.cell_1_enable"
*)

(* ===== HMI "HMI_RT_1" =====
system functions are stored by id; their names below are inferred from use

ScreenModuleEditorView "Row_Wire" 600x65
   Rectangle "Border" at 0,0 size 600x65
      Visibility <- "interface.background_visible"
      Appearance <- "interface.background_animate"
   TextField "TF R0 C0" at 5,5 size 360x60; Text 'CARBON WIRE'
      Visibility <- "interface.cell_0_visible"
   IOField "IOF R0 C1" at 370,5 size 225x60; FormatPattern 9999999
      on OnFinishInput: SetBit("interface.cell_1_input_finished")
      Visibility <- "interface.cell_1_visible"
      ObjectEnable <- "interface.cell_1_enable"
*)

(* ===== HMI "HMI_RT_1" =====
system functions are stored by id; their names below are inferred from use

ScreenModuleEditorView "Row_Wire" 600x65
   Rectangle "Border" at 0,0 size 600x65
      Visibility <- "interface.background_visible"
      Appearance <- "interface.background_animate"
   TextField "TF R0 C0" at 5,5 size 360x60; Text 'CARBON WIRE'
      Visibility <- "interface.cell_0_visible"
      Appearance <- "interface.cell_0_animate"
   IOField "IOF R0 C1" at 370,5 size 225x60; FormatPattern 9999999
      on OnFinishInput: SetBit("interface.cell_1_input_finished")
      Visibility <- "interface.cell_1_visible"
      ObjectEnable <- "interface.cell_1_enable"
      Appearance <- "interface.cell_1_animate"
*)

(* ===== HMI "HMI_RT_1" =====
system functions are stored by id; their names below are inferred from use

ScreenModuleEditorView "Row_Wire_Label" 600x65
   Rectangle "Border" at 0,0 size 600x65
      Visibility <- "interface.background_visible"
      Appearance <- "interface.background_animate"
   TextField "TF R0 C0" at 5,5 size 360x60; Text 'CARBON WIRE'
      Visibility <- "interface.cell_0_visible"
      Appearance <- "interface.cell_0_animate"
   IOField "IOF R0 C1" at 370,5 size 225x60; FormatPattern 9999999
      on OnFinishInput: SetBit("interface.cell_1_input_finished")
      Visibility <- "interface.cell_1_visible"
      Appearance <- "interface.cell_1_animate"
      ObjectEnable <- "interface.cell_1_enable"
*)

(* ===== HMI "HMI_RT_1" =====

ScreenModuleEditorView "Row_Wire_Label" 600x65
   Rectangle "Border" at 0,0 size 600x65
      Visibility <- "interface.background_visible"
      Appearance <- "interface.background_animate"
   TextField "TF R0 C0" at 5,5 size 360x60; Text 'WIRE'
      Visibility <- "interface.cell_0_visible"
      Appearance <- "interface.cell_0_animate"
   TextField "TF R0 C1" at 370,5 size 225x60; Text 'LENGTH'
      Visibility <- "interface.cell_1_visible"
      Appearance <- "interface.cell_1_animate"
*)

(* ===== HMI "HMI_RT_1" =====

ScreenModuleEditorView "Divider" 600x5
   Line "line" at 10,2 size 580x0
      Appearance <- "interface.line_animate"
      Visibility <- "interface.line_visible"
   Rectangle "background" at 0,0 size 600x5
      Appearance <- "interface.background_animate"
      Visibility <- "interface.background_visible"
*)

(* ===== HMI "HMI_RT_1" =====
system functions are stored by id; their names below are inferred from use

ScreenModuleEditorView "Navigation" 800x65
   Button "Wire" at 5,5 size 390x60; TextOff 'WIRE'
      Appearance <- "interface.wire_animate"
      on Press: function_b14e0dd5("interface.wire_actuate", 0)
   Button "Material" at 400,5 size 390x60; TextOff 'MATERIAL'
      Appearance <- "interface.material_animate"
      on Press: function_b14e0dd5("interface.material_actuate", 0)
   Rectangle "Wire_Cover" at 10,60 size 380x5
      Visibility <- "interface.wire_cover_visible"
   Rectangle "Material_Cover" at 405,60 size 380x5
      Visibility <- "interface.material_cover_visible"
*)

(* ===== HMI "HMI_RT_1" =====
system functions are stored by id; their names below are inferred from use

ScreenModuleEditorView "Navigation" 800x65
   Button "Wire" at 5,5 size 390x60; TextOff 'WIRE'
      on Press: function_b14e0dd5("interface.wire_actuate", 0)
      Appearance <- "interface.wire_animate"
   Button "Material" at 400,5 size 390x60; TextOff 'MATERIAL'
      on Press: function_b14e0dd5("interface.material_actuate", 0)
      Appearance <- "interface.material_animate"
   Rectangle "Wire_Cover" at 10,60 size 380x5
      Visibility <- "interface.wire_cover_visible"
   Rectangle "Material_Cover" at 405,60 size 380x5
      Visibility <- "interface.material_cover_visible"
*)

(* ===== HMI "HMI_RT_1" =====
system functions are stored by id; their names below are inferred from use

ScreenModuleEditorView "Navigation" 800x65
   Button "Wire" at 5,5 size 392x60; TextOff 'WIRE'
      on Press: function_b14e0dd5("interface.wire_actuate", 0)
      Appearance <- "interface.wire_animate"
   Button "Material" at 402,5 size 393x60; TextOff 'MATERIAL'
      on Press: function_b14e0dd5("interface.material_actuate", 0)
      Appearance <- "interface.material_animate"
   Rectangle "Wire_Cover" at 10,60 size 382x5
      Visibility <- "interface.wire_cover_visible"
   Rectangle "Material_Cover" at 407,60 size 383x5
      Visibility <- "interface.material_cover_visible"
*)

(* ===== HMI "HMI_RT_1" =====
system functions are stored by id; their names below are inferred from use

ScreenModuleEditorView "Row_Material" 600x65
   Rectangle "Border" at 0,0 size 600x65
      Visibility <- "interface.background_visible"
      Appearance <- "interface.background_animate"
   TextField "TF R0 C0" at 5,5 size 360x60; Text 'CARBON WIRE'
      Visibility <- "interface.cell_0_visible"
      Appearance <- "interface.cell_0_animate"
   IOField "IOF R0 C1" at 370,5 size 225x60; FormatPattern 9999999
      on OnFinishInput: SetBit("interface.cell_1_input_finished")
      Visibility <- "interface.cell_1_visible"
      Appearance <- "interface.cell_1_animate"
      ObjectEnable <- "interface.cell_1_enable"
*)

(* ===== HMI "HMI_RT_1" =====
system functions are stored by id; their names below are inferred from use

ScreenModuleEditorView "Row_Material" 600x40
   Rectangle "Border" at 0,0 size 600x40
      Visibility <- "interface.background_visible"
      Appearance <- "interface.background_animate"
   IOField "IOF R0 C1" at 370,5 size 225x35; FormatPattern 9999999
      on OnFinishInput: SetBit("interface.cell_1_input_finished")
      Visibility <- "interface.cell_1_visible"
      Appearance <- "interface.cell_1_animate"
      ObjectEnable <- "interface.cell_1_enable"
   TextField "TF R0 C0" at 5,5 size 360x35; Text 'MOLYBDENUM'
      Visibility <- "interface.cell_0_visible"
      Appearance <- "interface.cell_0_animate"
*)

(* ===== HMI "HMI_RT_1" =====
system functions are stored by id; their names below are inferred from use

ScreenModuleEditorView "Row_Custom" 600x40
   Rectangle "Border" at 0,0 size 600x40
      Visibility <- "interface.background_visible"
      Appearance <- "interface.background_animate"
   IOField "IOF R0 C1" at 370,5 size 225x35; FormatPattern 9999999
      on OnFinishInput: SetBit("interface.cell_1_input_finished")
      Visibility <- "interface.cell_1_visible"
      Appearance <- "interface.cell_1_animate"
      ObjectEnable <- "interface.cell_1_enable"
   TextField "TF R0 C0" at 5,5 size 360x35; Text 'MOLYBDENUM'
      Visibility <- "interface.cell_0_visible"
      Appearance <- "interface.cell_0_animate"
*)

(* ===== HMI "HMI_RT_1" =====
system functions are stored by id; their names below are inferred from use

ScreenModuleEditorView "Row_Custom" 600x40
   Rectangle "Border" at 0,0 size 600x40
      Visibility <- "interface.background_visible"
      Appearance <- "interface.background_animate"
   IOField "IOF R0 C0" at 5,5 size 360x35; FormatPattern ???????????????
      on OnFinishInput: SetBit("interface.cell_0_input_finished")
      Appearance <- "interface.cell_0_animate"
      ObjectEnable <- "interface.cell_0_enable"
      Visibility <- "interface.cell_0_visible"
   IOField "IOF R0 C1" at 370,5 size 225x35; FormatPattern 9999999
      on OnFinishInput: SetBit("interface.cell_1_input_finished")
      Visibility <- "interface.cell_1_visible"
      Appearance <- "interface.cell_1_animate"
      ObjectEnable <- "interface.cell_1_enable"
*)

(* ===== HMI "HMI_RT_1" =====
system functions are stored by id; their names below are inferred from use

ScreenModuleEditorView "Row_Material_Label" 600x40
   Rectangle "Border" at 0,0 size 600x40
      Visibility <- "interface.background_visible"
      Appearance <- "interface.background_animate"
   IOField "IOF R0 C1" at 370,5 size 225x35; FormatPattern 9999999
      on OnFinishInput: SetBit("interface.cell_1_input_finished")
      Visibility <- "interface.cell_1_visible"
      Appearance <- "interface.cell_1_animate"
      ObjectEnable <- "interface.cell_1_enable"
   TextField "TF R0 C0" at 5,5 size 360x35; Text 'MOLYBDENUM'
      Visibility <- "interface.cell_0_visible"
      Appearance <- "interface.cell_0_animate"
*)

(* ===== HMI "HMI_RT_1" =====

ScreenModuleEditorView "Row_Material_Label" 600x40
   Rectangle "Border" at 0,0 size 600x40
      Visibility <- "interface.background_visible"
      Appearance <- "interface.background_animate"
   TextField "TF R0 C0" at 5,5 size 360x35; Text 'MATERIAL'
      Visibility <- "interface.cell_0_visible"
      Appearance <- "interface.cell_0_animate"
   TextField "TF R0 C1" at 370,5 size 225x35; Text 'BAGS'
      Appearance <- "interface.cell_1_animate"
      Visibility <- "interface.cell_1_visible"
*)

(* ===== HMI "HMI_RT_1" =====
system functions are stored by id; their names below are inferred from use

ScreenModuleEditorView "Row_Wire" 600x65
   Rectangle "Border" at 0,0 size 600x65
      Visibility <- "interface.background_visible"
   TextField "TF R0 C0" at 5,5 size 360x60; Text 'CARBON WIRE'
      Visibility <- "interface.cell_0_visible"
   IOField "IOF R0 C1" at 370,5 size 225x60; FormatPattern 9999999
      on OnFinishInput: SetBit("interface.cell_1_input_finished")
      Visibility <- "interface.cell_1_visible"
      Appearance <- "interface.cell_1_animate"
      ObjectEnable <- "interface.cell_1_enable"
*)